PROGRAM Anlage
VAR_INPUT
	UR5				:FB_Roboter;
	Gripper			:FB_SmartGreifer;
	HEX_E			:FB_Kraftsensor; 
END_VAR

VAR
END_VAR

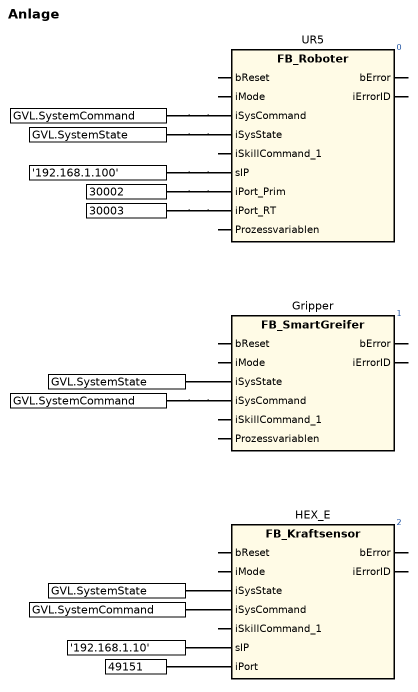
UR5(
    iSysCommand := GVL.SystemCommand,
    iSysState := GVL.SystemState,
    sIP := '192.168.1.100',
    iPort_Prim := 30002,
    iPort_RT := 30003); // FB_Roboter
Gripper(iSysState := GVL.SystemState, iSysCommand := GVL.SystemCommand); // FB_SmartGreifer
HEX_E(iSysState := GVL.SystemState, iSysCommand := GVL.SystemCommand, sIP := '192.168.1.10', iPort := 49151); // FB_Kraftsensor

END_PROGRAM

(* stored: Version 1.1.0.1
   POU Anlage: Id {ff8182a3-48a3-4c02-a4af-58fad1227f8f}, SpecialFunc None *)
